(* Logix 5000 project; controller MainProject_v1 1756-L85E rev 36.11; software revision 36.00 *)

TASK MainTask (continuous, watchdog 500 ms) : MainProgram

MODULES
   Local : 1756-L85E (ICP 0, rev 36.11)
END_MODULES

VAR_GLOBAL   (* controller tags *)
   Dharmendra : STRING;
   DT1 : TIMER := (PRE := 10000);
   Inp_FromLDSDK : DINT;
   on1 : BOOL;
   RUN1 : BOOL;
   sd : STRING;
   Start : BOOL;
   start1 : BOOL;
   start11 : BOOL;
   STOP1 : BOOL;
   test : TIMER := (PRE := 1000);
   Val_Seconds : DINT;
END_VAR

PROGRAM MainProgram   (* main routine MainRoutine *)
VAR
   TON_1Second : TIMER := (PRE := 1000);
END_VAR

ROUTINE MainRoutine   (* ladder *)
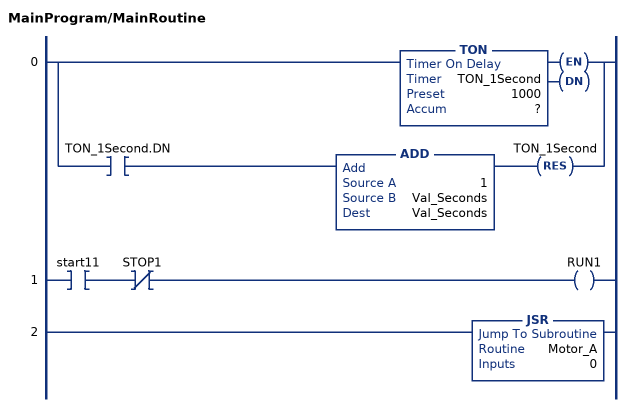
   0: [TON(TON_1Second,?,?) ,XIC(TON_1Second.DN) ADD(1,Val_Seconds,Val_Seconds) RES(TON_1Second) ];
   1: XIC(start11)XIO(STOP1)OTE(RUN1);
   2: JSR(Motor_A,0);
END_ROUTINE

ROUTINE Motor_A   (* ladder *)
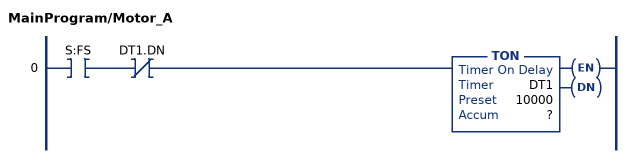
   0: XIC(S:FS)XIO(DT1.DN)TON(DT1,?,?);
END_ROUTINE
END_PROGRAM
